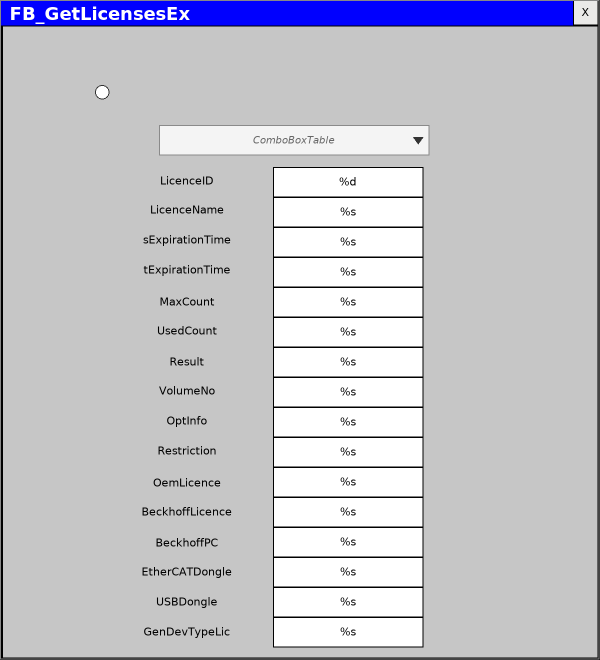
VISUALIZATION dialogGetLicensesEx  // 600x660
    Rectangle (0,0 600x660)
        OnMouseClick: CloseDialog Dialog=dialogGetLicensesEx, Result=OK, NumpadKeypadSet=True
    Rectangle (0,0 600x26), "FB_GetLicensesEx"
    Rectangle (573,0 25x25), "X"
        OnMouseClick: CloseDialog Dialog=dialogReject, Result=Cancel, NumpadKeypadSet=True
    Rectangle (273,167 150x30), "%d", text variable: System.tActiveLicenceArray.stLicenseId
    Label (112,166 150x30), "LicenceID"
    Label (112,195 150x30), "LicenceName"
    Rectangle (273,197 150x30), "%s", text variable: System.tActiveLicenceArray.sLicenseName
    Label (112,225 150x30), "sExpirationTime"
    Rectangle (273,227 150x30), "%s", text variable: System.tActiveLicenceArray.sExpirationTime
    Label (112,255 150x30), "tExpirationTime"
    Rectangle (273,257 150x30), "%s", text variable: System.tActiveLicenceArray.tExpirationTime
    Label (112,287 150x30), "MaxCount"
    Rectangle (273,287 150x30), "%s", text variable: System.tActiveLicenceArray.nMaxCount
    Label (112,316 150x30), "UsedCount"
    Rectangle (273,317 150x30), "%s", text variable: System.tActiveLicenceArray.nUsedCount
    Rectangle (273,347 150x30), "%s", text variable: System.tActiveLicenceArray.eResult
    Label (112,347 150x30), "Result"
    Label (112,376 150x30), "VolumeNo"
    Rectangle (273,377 150x30), "%s", text variable: System.tActiveLicenceArray.nVolumeNo
    Label (112,406 150x30), "OptInfo"
    Rectangle (273,407 150x30), "%s", text variable: System.tActiveLicenceArray.nOptInfo
    Label (112,436 150x30), "Restriction"
    Rectangle (273,437 150x30), "%s", text variable: System.tActiveLicenceArray.nRestriction
    Label (112,468 150x30), "OemLicence"
    Rectangle (273,467 150x30), "%s", text variable: System.tActiveLicenceArray.bOemLicense
    Label (112,497 150x30), "BeckhoffLicence"
    Rectangle (273,497 150x30), "%s", text variable: System.tActiveLicenceArray.bBeckhoffLicense
    Rectangle (273,527 150x30), "%s", text variable: System.tActiveLicenceArray.bBeckhoffPC
    Label (112,528 150x30), "BeckhoffPC"
    Label (112,557 150x30), "EtherCATDongle"
    Rectangle (273,557 150x30), "%s", text variable: System.tActiveLicenceArray.bEtherCATDongle
    Label (112,587 150x30), "USBDongle"
    Rectangle (273,587 150x30), "%s", text variable: System.tActiveLicenceArray.bUSBDongle
    Label (112,617 150x30), "GenDevTypeLic"
    Rectangle (273,617 150x30), "%s", text variable: System.tActiveLicenceArray.bGenDevTypeLic
    RadioButton (93,37 454x110), variable: System.licenceType
        Areas[0]: Text=Valid Licences
        Areas[1]: Text=Pending Licences
        Areas[2]: Text=Demo Licences
        Areas[3]: Text=OEM Licences
        Areas[4]: Text=Failed Licences
        Areas[5]: Text=Invalid Licences
    ComboBoxTable (159,125 270x30), variable: System.tActiveLicenceSel, data array: System.tActiveLicenceList
        p1892666644: System.tActiveLicenceArray.sLicenseName
        p338671338: System.tActiveLicenceArray.tExpirationTime
        p2170511999: System.tActiveLicenceArray.sExpirationTime
        p3723444502: System.tActiveLicenceArray.nMaxCount
        p1218418051: System.tActiveLicenceArray.nUsedCount
        p746581629: System.tActiveLicenceArray.eResult
        p3104783080: System.tActiveLicenceArray.nVolumeNo
        p2501879983: System.tActiveLicenceArray.nOptInfo
        p7306298: System.tActiveLicenceArray.nRestriction
        p1933151965: System.tActiveLicenceArray.bOemLicense
        p3863566920: System.tActiveLicenceArray.bBeckhoffLicense
        p2192122294: System.tActiveLicenceArray.bBeckhoffPC
        p400160035: System.tActiveLicenceArray.bEtherCATDongle
        p1265227338: System.tActiveLicenceArray.bUSBDongle
        p3726181087: System.tActiveLicenceArray.bGenDevTypeLic
        p3854506369: System.tActiveLicenceList[INDEX]
END_VISUALIZATION

(* stored: Version 1.1.0.1, ProductVersion 3.1.4024.12
   Visu dialogGetLicensesEx: Id {69f871ba-beb8-4d61-b141-52f30c3098b8} *)
